// Mitsubishi GX Works2 project: pr3   PLC: Q03UDV

PROGRAM MAIN
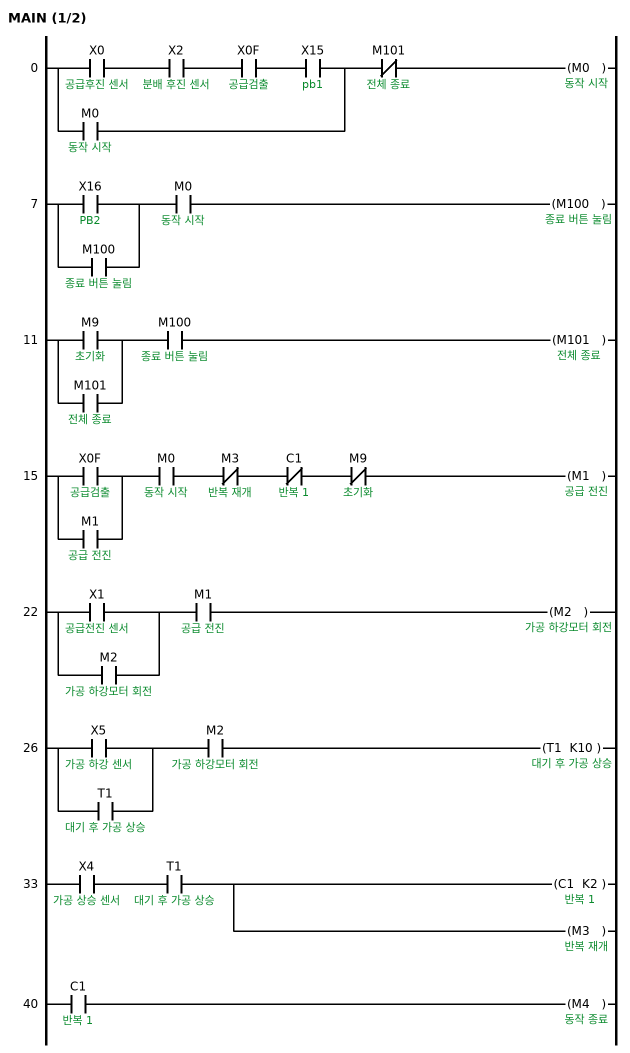
0     LD      X0  ; 공급후진 센서
      AND     X2  ; 분배 후진 센서
      AND     X0F  ; 공급검출
      AND     X15  ; pb1
      OR      M0  ; 동작 시작
      ANI     M101  ; 전체 종료
      OUT     M0  ; 동작 시작
7     LD      X16  ; PB2
      OR      M100  ; 종료 버튼 눌림
      AND     M0  ; 동작 시작
      OUT     M100  ; 종료 버튼 눌림
11    LD      M9  ; 초기화
      OR      M101  ; 전체 종료
      AND     M100  ; 종료 버튼 눌림
      OUT     M101  ; 전체 종료
15    LD      X0F  ; 공급검출
      OR      M1  ; 공급 전진
      AND     M0  ; 동작 시작
      ANI     M3  ; 반복 재개
      ANI     C1  ; 반복 1
      ANI     M9  ; 초기화
      OUT     M1  ; 공급 전진
22    LD      X1  ; 공급전진 센서
      OR      M2  ; 가공 하강모터 회전
      AND     M1  ; 공급 전진
      OUT     M2  ; 가공 하강모터 회전
26    LD      X5  ; 가공 하강 센서
      OR      T1  ; 대기 후 가공 상승
      AND     M2  ; 가공 하강모터 회전
      OUT     T1 K10  ; 대기 후 가공 상승
33    LD      X4  ; 가공 상승 센서
      AND     T1  ; 대기 후 가공 상승
      OUT     C1 K2  ; 반복 1
      OUT     M3  ; 반복 재개
40    LD      C1  ; 반복 1
      OUT     M4  ; 동작 종료
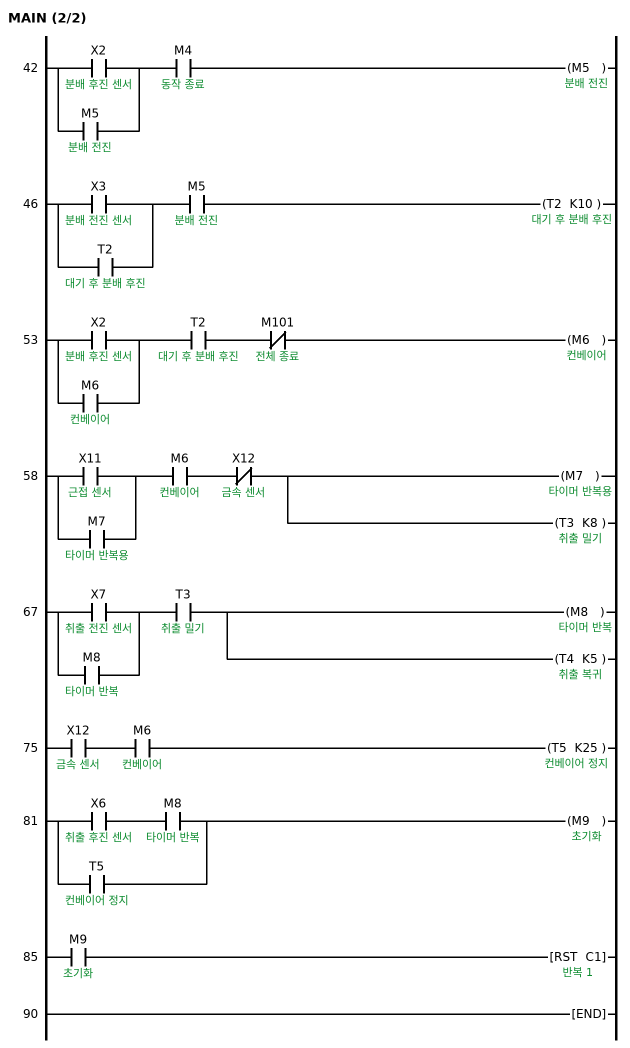
42    LD      X2  ; 분배 후진 센서
      OR      M5  ; 분배 전진
      AND     M4  ; 동작 종료
      OUT     M5  ; 분배 전진
46    LD      X3  ; 분배 전진 센서
      OR      T2  ; 대기 후 분배 후진
      AND     M5  ; 분배 전진
      OUT     T2 K10  ; 대기 후 분배 후진
53    LD      X2  ; 분배 후진 센서
      OR      M6  ; 컨베이어
      AND     T2  ; 대기 후 분배 후진
      ANI     M101  ; 전체 종료
      OUT     M6  ; 컨베이어
58    LD      X11  ; 근접 센서
      OR      M7  ; 타이머 반복용
      AND     M6  ; 컨베이어
      ANI     X12  ; 금속 센서
      OUT     M7  ; 타이머 반복용
      OUT     T3 K8  ; 취출 밀기
67    LD      X7  ; 취출 전진 센서
      OR      M8  ; 타이머 반복
      AND     T3  ; 취출 밀기
      OUT     M8  ; 타이머 반복
      OUT     T4 K5  ; 취출 복귀
75    LD      X12  ; 금속 센서
      AND     M6  ; 컨베이어
      OUT     T5 K25  ; 컨베이어 정지
81    LD      X6  ; 취출 후진 센서
      AND     M8  ; 타이머 반복
      OR      T5  ; 컨베이어 정지
      OUT     M9  ; 초기화
85    LD      M9  ; 초기화
      RST     C1  ; 반복 1
90    END
END_PROGRAM

PROGRAM OUTPUT
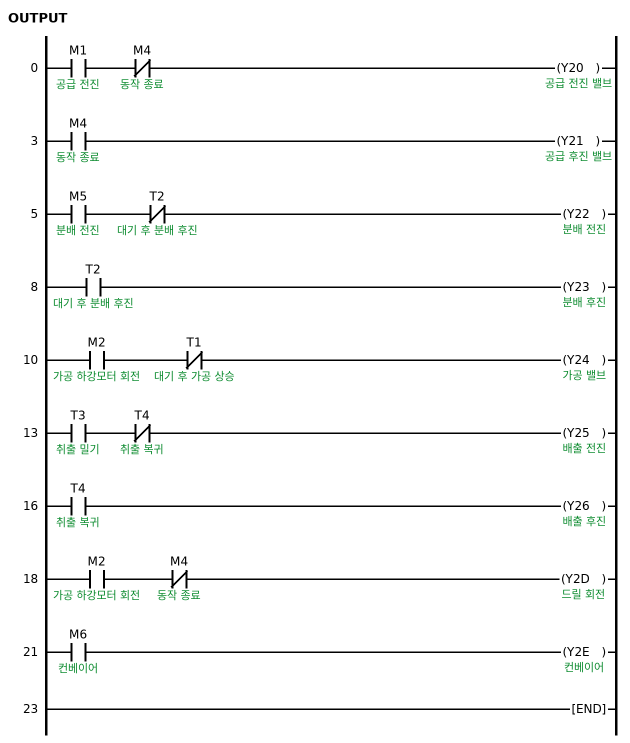
0     LD      M1  ; 공급 전진
      ANI     M4  ; 동작 종료
      OUT     Y20  ; 공급 전진 밸브
3     LD      M4  ; 동작 종료
      OUT     Y21  ; 공급 후진 밸브
5     LD      M5  ; 분배 전진
      ANI     T2  ; 대기 후 분배 후진
      OUT     Y22  ; 분배 전진
8     LD      T2  ; 대기 후 분배 후진
      OUT     Y23  ; 분배 후진
10    LD      M2  ; 가공 하강모터 회전
      ANI     T1  ; 대기 후 가공 상승
      OUT     Y24  ; 가공 밸브
13    LD      T3  ; 취출 밀기
      ANI     T4  ; 취출 복귀
      OUT     Y25  ; 배출 전진
16    LD      T4  ; 취출 복귀
      OUT     Y26  ; 배출 후진
18    LD      M2  ; 가공 하강모터 회전
      ANI     M4  ; 동작 종료
      OUT     Y2D  ; 드릴 회전
21    LD      M6  ; 컨베이어
      OUT     Y2E  ; 컨베이어
23    END
END_PROGRAM

// device comments not shown above
X10  ; 근접 센서
